FUNCTION CheckDivDWord : DWORD
VAR_INPUT
	divisor				: DWORD;
END_VAR
VAR
END_VAR

IF divisor = 0 THEN
	CheckDWordZeroDiv_ErrCnt := CheckDWordZeroDiv_ErrCnt + 1;
	CheckDivDWord := 1;
ELSE
	CheckDivDWord := divisor;
END_IF

END_FUNCTION

(* stored: Version 1.1.0.1, ProductVersion 3.1.4024.12
   POU CheckDivDWord: Id {76b02a87-804a-4b6a-924a-acd947610302}, SpecialFunc CheckDivInt64 *)
